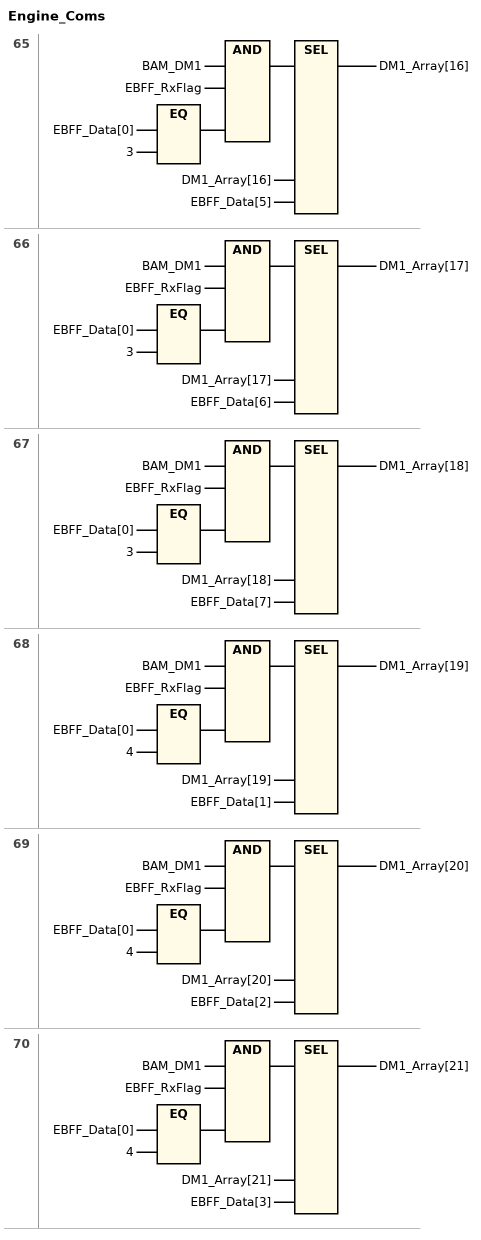
// NETWORK 65
DM1_Array[16] := SEL(BAM_DM1 AND EBFF_RxFlag AND EBFF_Data[0] = 3, DM1_Array[16], EBFF_Data[5]);

// NETWORK 66
DM1_Array[17] := SEL(BAM_DM1 AND EBFF_RxFlag AND EBFF_Data[0] = 3, DM1_Array[17], EBFF_Data[6]);

// NETWORK 67
DM1_Array[18] := SEL(BAM_DM1 AND EBFF_RxFlag AND EBFF_Data[0] = 3, DM1_Array[18], EBFF_Data[7]);

// NETWORK 68
DM1_Array[19] := SEL(BAM_DM1 AND EBFF_RxFlag AND EBFF_Data[0] = 4, DM1_Array[19], EBFF_Data[1]);

// NETWORK 69
DM1_Array[20] := SEL(BAM_DM1 AND EBFF_RxFlag AND EBFF_Data[0] = 4, DM1_Array[20], EBFF_Data[2]);

// NETWORK 70
DM1_Array[21] := SEL(BAM_DM1 AND EBFF_RxFlag AND EBFF_Data[0] = 4, DM1_Array[21], EBFF_Data[3]);

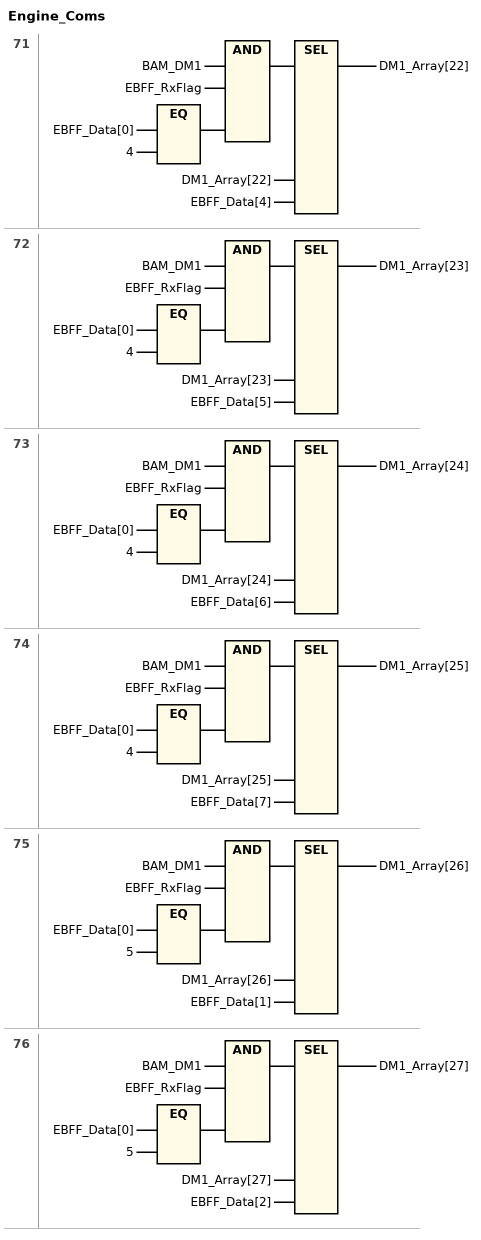
// NETWORK 71
DM1_Array[22] := SEL(BAM_DM1 AND EBFF_RxFlag AND EBFF_Data[0] = 4, DM1_Array[22], EBFF_Data[4]);

// NETWORK 72
DM1_Array[23] := SEL(BAM_DM1 AND EBFF_RxFlag AND EBFF_Data[0] = 4, DM1_Array[23], EBFF_Data[5]);

// NETWORK 73
DM1_Array[24] := SEL(BAM_DM1 AND EBFF_RxFlag AND EBFF_Data[0] = 4, DM1_Array[24], EBFF_Data[6]);

// NETWORK 74
DM1_Array[25] := SEL(BAM_DM1 AND EBFF_RxFlag AND EBFF_Data[0] = 4, DM1_Array[25], EBFF_Data[7]);

// NETWORK 75
DM1_Array[26] := SEL(BAM_DM1 AND EBFF_RxFlag AND EBFF_Data[0] = 5, DM1_Array[26], EBFF_Data[1]);

// NETWORK 76
DM1_Array[27] := SEL(BAM_DM1 AND EBFF_RxFlag AND EBFF_Data[0] = 5, DM1_Array[27], EBFF_Data[2]);

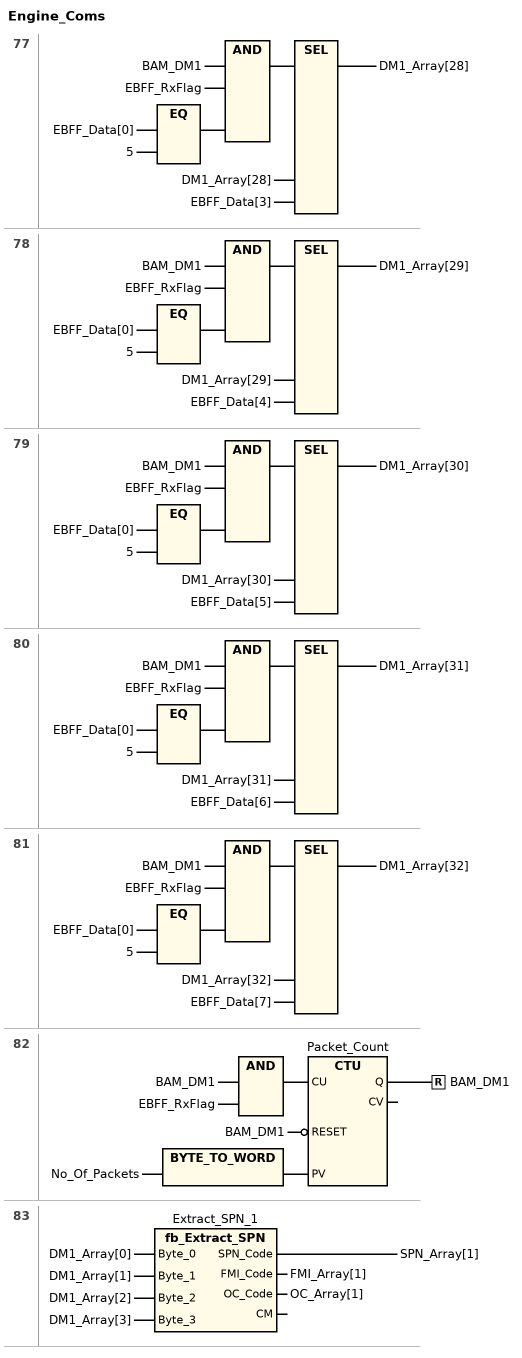
// NETWORK 77
DM1_Array[28] := SEL(BAM_DM1 AND EBFF_RxFlag AND EBFF_Data[0] = 5, DM1_Array[28], EBFF_Data[3]);

// NETWORK 78
DM1_Array[29] := SEL(BAM_DM1 AND EBFF_RxFlag AND EBFF_Data[0] = 5, DM1_Array[29], EBFF_Data[4]);

// NETWORK 79
DM1_Array[30] := SEL(BAM_DM1 AND EBFF_RxFlag AND EBFF_Data[0] = 5, DM1_Array[30], EBFF_Data[5]);

// NETWORK 80
DM1_Array[31] := SEL(BAM_DM1 AND EBFF_RxFlag AND EBFF_Data[0] = 5, DM1_Array[31], EBFF_Data[6]);

// NETWORK 81
DM1_Array[32] := SEL(BAM_DM1 AND EBFF_RxFlag AND EBFF_Data[0] = 5, DM1_Array[32], EBFF_Data[7]);

// NETWORK 82
Packet_Count(CU := BAM_DM1 AND EBFF_RxFlag, RESET := NOT BAM_DM1, PV := BYTE_TO_WORD(No_Of_Packets)); // CTU
BAM_DM1 R= Packet_Count.Q;

// NETWORK 83
Extract_SPN_1(
    Byte_0 := DM1_Array[0],
    Byte_1 := DM1_Array[1],
    Byte_2 := DM1_Array[2],
    Byte_3 := DM1_Array[3],
    FMI_Code => FMI_Array[1],
    OC_Code => OC_Array[1]); // fb_Extract_SPN
SPN_Array[1] := Extract_SPN_1.SPN_Code;

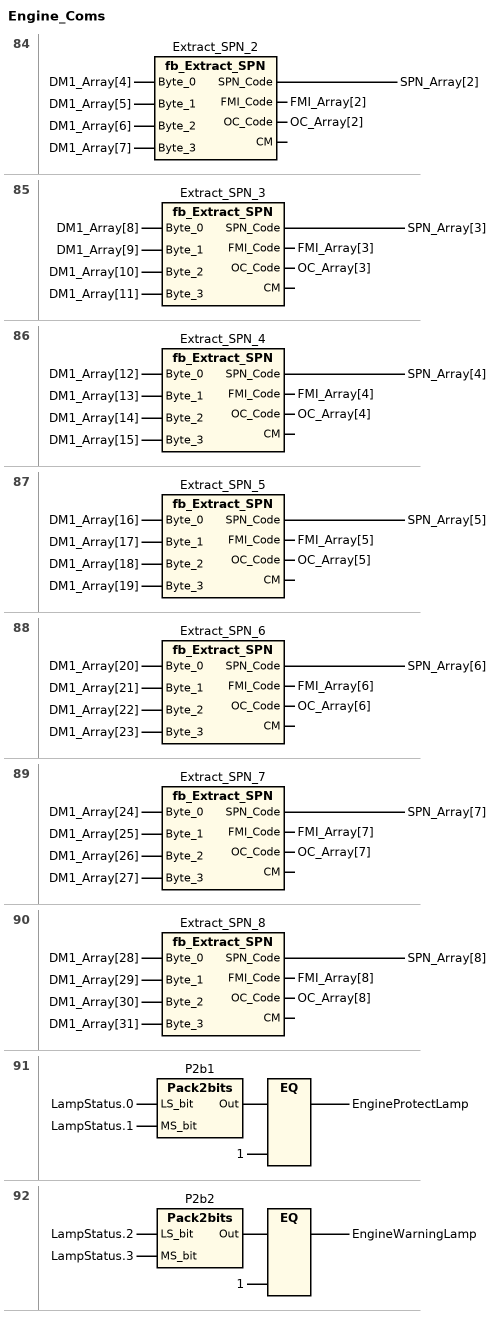
// NETWORK 84
Extract_SPN_2(
    Byte_0 := DM1_Array[4],
    Byte_1 := DM1_Array[5],
    Byte_2 := DM1_Array[6],
    Byte_3 := DM1_Array[7],
    FMI_Code => FMI_Array[2],
    OC_Code => OC_Array[2]); // fb_Extract_SPN
SPN_Array[2] := Extract_SPN_2.SPN_Code;

// NETWORK 85
Extract_SPN_3(
    Byte_0 := DM1_Array[8],
    Byte_1 := DM1_Array[9],
    Byte_2 := DM1_Array[10],
    Byte_3 := DM1_Array[11],
    FMI_Code => FMI_Array[3],
    OC_Code => OC_Array[3]); // fb_Extract_SPN
SPN_Array[3] := Extract_SPN_3.SPN_Code;

// NETWORK 86
Extract_SPN_4(
    Byte_0 := DM1_Array[12],
    Byte_1 := DM1_Array[13],
    Byte_2 := DM1_Array[14],
    Byte_3 := DM1_Array[15],
    FMI_Code => FMI_Array[4],
    OC_Code => OC_Array[4]); // fb_Extract_SPN
SPN_Array[4] := Extract_SPN_4.SPN_Code;

// NETWORK 87
Extract_SPN_5(
    Byte_0 := DM1_Array[16],
    Byte_1 := DM1_Array[17],
    Byte_2 := DM1_Array[18],
    Byte_3 := DM1_Array[19],
    FMI_Code => FMI_Array[5],
    OC_Code => OC_Array[5]); // fb_Extract_SPN
SPN_Array[5] := Extract_SPN_5.SPN_Code;

// NETWORK 88
Extract_SPN_6(
    Byte_0 := DM1_Array[20],
    Byte_1 := DM1_Array[21],
    Byte_2 := DM1_Array[22],
    Byte_3 := DM1_Array[23],
    FMI_Code => FMI_Array[6],
    OC_Code => OC_Array[6]); // fb_Extract_SPN
SPN_Array[6] := Extract_SPN_6.SPN_Code;

// NETWORK 89
Extract_SPN_7(
    Byte_0 := DM1_Array[24],
    Byte_1 := DM1_Array[25],
    Byte_2 := DM1_Array[26],
    Byte_3 := DM1_Array[27],
    FMI_Code => FMI_Array[7],
    OC_Code => OC_Array[7]); // fb_Extract_SPN
SPN_Array[7] := Extract_SPN_7.SPN_Code;

// NETWORK 90
Extract_SPN_8(
    Byte_0 := DM1_Array[28],
    Byte_1 := DM1_Array[29],
    Byte_2 := DM1_Array[30],
    Byte_3 := DM1_Array[31],
    FMI_Code => FMI_Array[8],
    OC_Code => OC_Array[8]); // fb_Extract_SPN
SPN_Array[8] := Extract_SPN_8.SPN_Code;

// NETWORK 91
P2b1(LS_bit := LampStatus.0, MS_bit := LampStatus.1); // Pack2bits
EngineProtectLamp := P2b1.Out = 1;

// NETWORK 92
P2b2(LS_bit := LampStatus.2, MS_bit := LampStatus.3); // Pack2bits
EngineWarningLamp := P2b2.Out = 1;

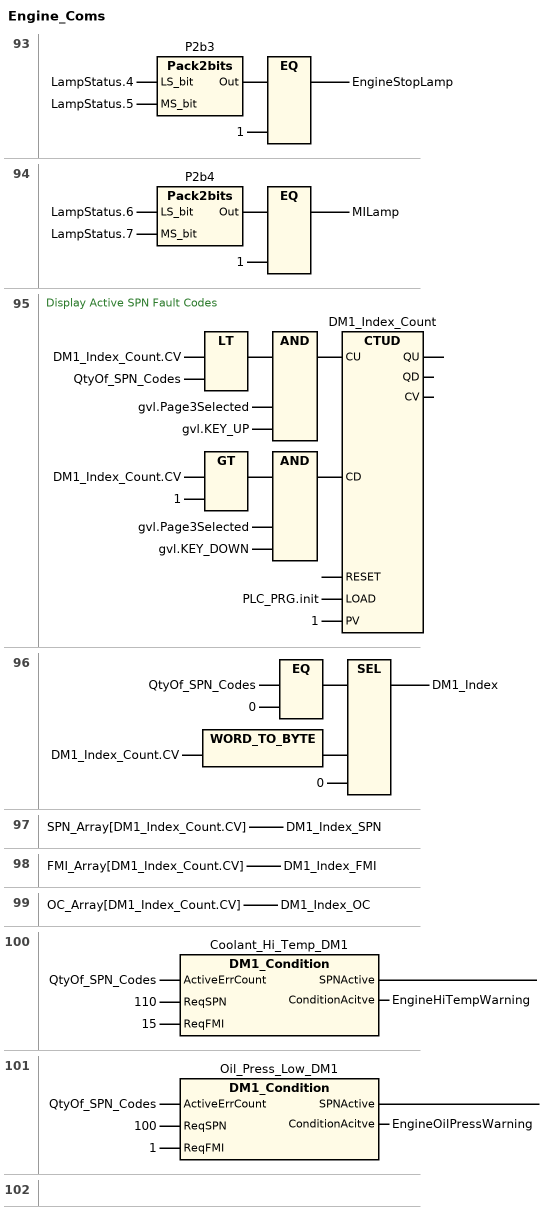
// NETWORK 93
P2b3(LS_bit := LampStatus.4, MS_bit := LampStatus.5); // Pack2bits
EngineStopLamp := P2b3.Out = 1;

// NETWORK 94
P2b4(LS_bit := LampStatus.6, MS_bit := LampStatus.7); // Pack2bits
MILamp := P2b4.Out = 1;

// NETWORK 95
// Display Active SPN Fault Codes
DM1_Index_Count(
    CU := DM1_Index_Count.CV < QtyOf_SPN_Codes AND gvl.Page3Selected AND gvl.KEY_UP,
    CD := DM1_Index_Count.CV > 1 AND gvl.Page3Selected AND gvl.KEY_DOWN,
    LOAD := PLC_PRG.init,
    PV := 1); // CTUD

// NETWORK 96
DM1_Index := SEL(QtyOf_SPN_Codes = 0, WORD_TO_BYTE(DM1_Index_Count.CV), 0);

// NETWORK 97
DM1_Index_SPN := SPN_Array[DM1_Index_Count.CV];

// NETWORK 98
DM1_Index_FMI := FMI_Array[DM1_Index_Count.CV];

// NETWORK 99
DM1_Index_OC := OC_Array[DM1_Index_Count.CV];

// NETWORK 100
Coolant_Hi_Temp_DM1(
    ActiveErrCount := QtyOf_SPN_Codes,
    ReqSPN := 110,
    ReqFMI := 15,
    ConditionAcitve => EngineHiTempWarning); // DM1_Condition

// NETWORK 101
Oil_Press_Low_DM1(
    ActiveErrCount := QtyOf_SPN_Codes,
    ReqSPN := 100,
    ReqFMI := 1,
    ConditionAcitve => EngineOilPressWarning); // DM1_Condition

// NETWORK 102

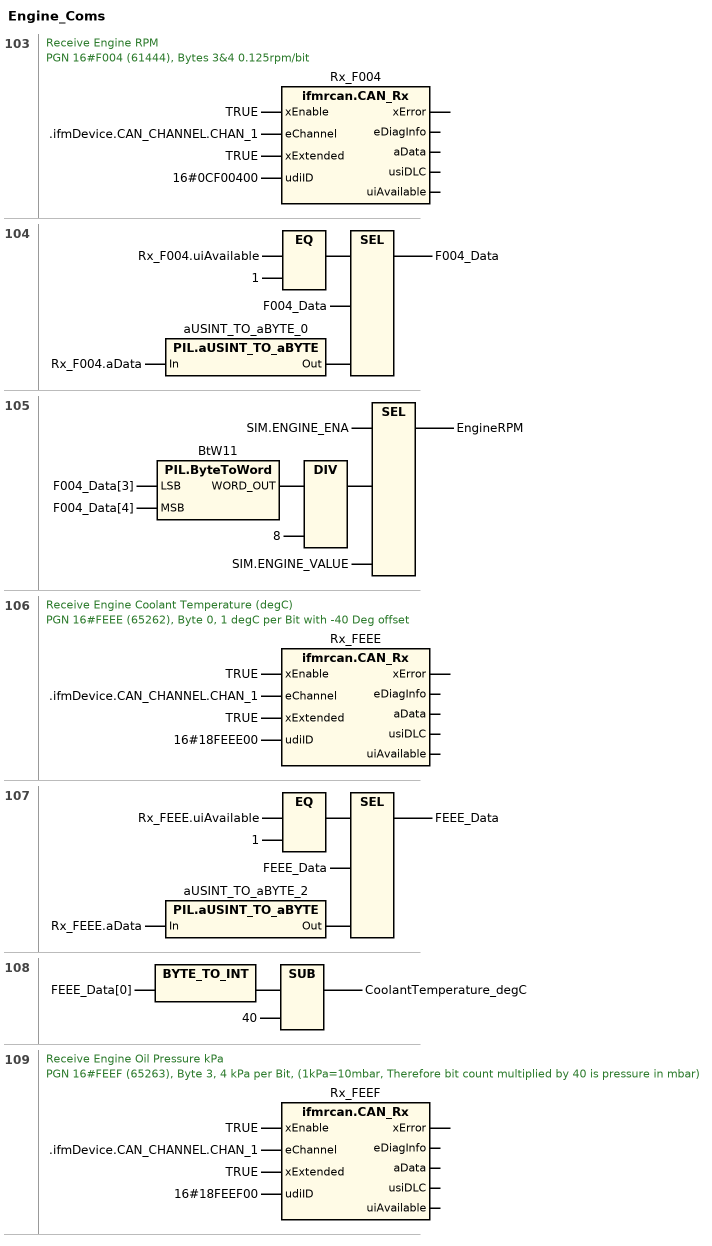
// NETWORK 103
// Receive Engine RPM
// PGN 16#F004 (61444), Bytes 3&4 0.125rpm/bit
Rx_F004(xEnable := TRUE, eChannel := .ifmDevice.CAN_CHANNEL.CHAN_1, xExtended := TRUE, udiID := 16#0CF00400); // ifmrcan.CAN_Rx

// NETWORK 104
aUSINT_TO_aBYTE_0(In := Rx_F004.aData); // PIL.aUSINT_TO_aBYTE
F004_Data := SEL(Rx_F004.uiAvailable = 1, F004_Data, aUSINT_TO_aBYTE_0.Out);

// NETWORK 105
BtW11(LSB := F004_Data[3], MSB := F004_Data[4]); // PIL.ByteToWord
EngineRPM := SEL(SIM.ENGINE_ENA, BtW11.WORD_OUT / 8, SIM.ENGINE_VALUE);

// NETWORK 106
// Receive Engine Coolant Temperature (degC)
// PGN 16#FEEE (65262), Byte 0, 1 degC per Bit with -40 Deg offset
Rx_FEEE(xEnable := TRUE, eChannel := .ifmDevice.CAN_CHANNEL.CHAN_1, xExtended := TRUE, udiID := 16#18FEEE00); // ifmrcan.CAN_Rx

// NETWORK 107
aUSINT_TO_aBYTE_2(In := Rx_FEEE.aData); // PIL.aUSINT_TO_aBYTE
FEEE_Data := SEL(Rx_FEEE.uiAvailable = 1, FEEE_Data, aUSINT_TO_aBYTE_2.Out);

// NETWORK 108
CoolantTemperature_degC := BYTE_TO_INT(FEEE_Data[0]) - 40;

// NETWORK 109
// Receive Engine Oil Pressure kPa
// PGN 16#FEEF (65263), Byte 3, 4 kPa per Bit, (1kPa=10mbar, Therefore bit count multiplied by 40 is pressure in mbar)
Rx_FEEF(xEnable := TRUE, eChannel := .ifmDevice.CAN_CHANNEL.CHAN_1, xExtended := TRUE, udiID := 16#18FEEF00); // ifmrcan.CAN_Rx

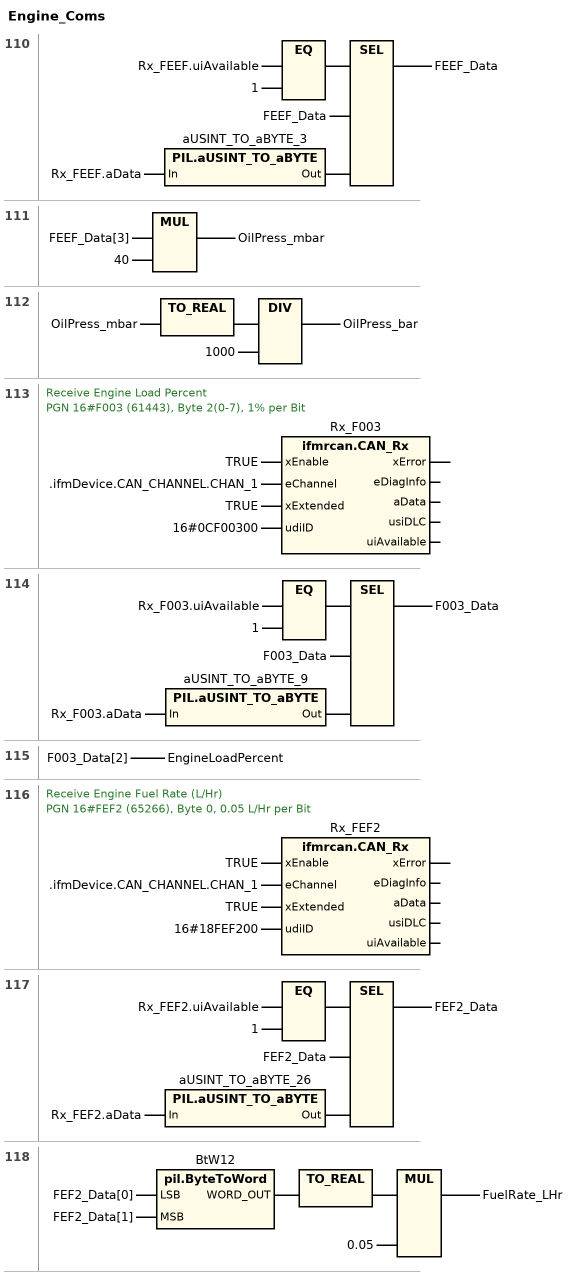
// NETWORK 110
aUSINT_TO_aBYTE_3(In := Rx_FEEF.aData); // PIL.aUSINT_TO_aBYTE
FEEF_Data := SEL(Rx_FEEF.uiAvailable = 1, FEEF_Data, aUSINT_TO_aBYTE_3.Out);

// NETWORK 111
OilPress_mbar := FEEF_Data[3] * 40;

// NETWORK 112
OilPress_bar := TO_REAL(OilPress_mbar) / 1000;

// NETWORK 113
// Receive Engine Load Percent
// PGN 16#F003 (61443), Byte 2(0-7), 1% per Bit
Rx_F003(xEnable := TRUE, eChannel := .ifmDevice.CAN_CHANNEL.CHAN_1, xExtended := TRUE, udiID := 16#0CF00300); // ifmrcan.CAN_Rx

// NETWORK 114
aUSINT_TO_aBYTE_9(In := Rx_F003.aData); // PIL.aUSINT_TO_aBYTE
F003_Data := SEL(Rx_F003.uiAvailable = 1, F003_Data, aUSINT_TO_aBYTE_9.Out);

// NETWORK 115
EngineLoadPercent := F003_Data[2];

// NETWORK 116
// Receive Engine Fuel Rate (L/Hr)
// PGN 16#FEF2 (65266), Byte 0, 0.05 L/Hr per Bit
Rx_FEF2(xEnable := TRUE, eChannel := .ifmDevice.CAN_CHANNEL.CHAN_1, xExtended := TRUE, udiID := 16#18FEF200); // ifmrcan.CAN_Rx

// NETWORK 117
aUSINT_TO_aBYTE_26(In := Rx_FEF2.aData); // PIL.aUSINT_TO_aBYTE
FEF2_Data := SEL(Rx_FEF2.uiAvailable = 1, FEF2_Data, aUSINT_TO_aBYTE_26.Out);

// NETWORK 118
BtW12(LSB := FEF2_Data[0], MSB := FEF2_Data[1]); // pil.ByteToWord
FuelRate_LHr := TO_REAL(BtW12.WORD_OUT) * 0.05;

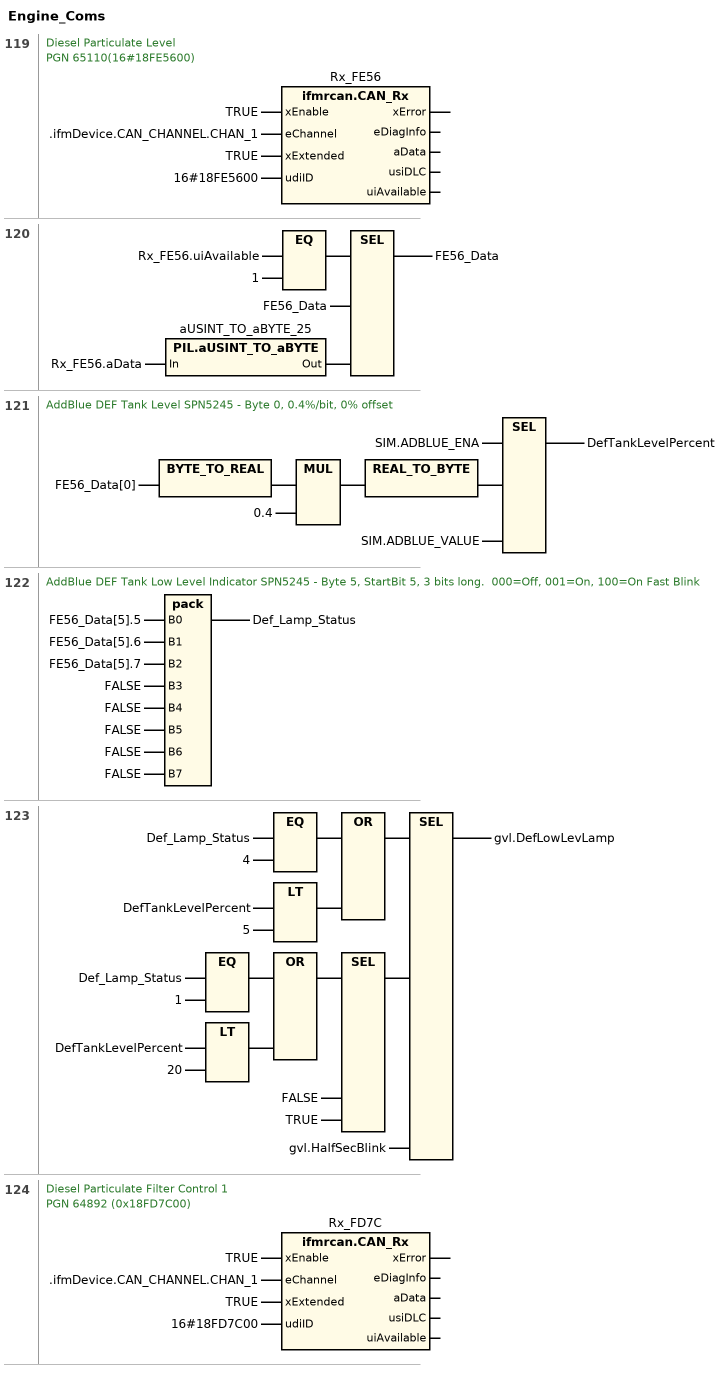
// NETWORK 119
// Diesel Particulate Level
// PGN 65110(16#18FE5600)
Rx_FE56(xEnable := TRUE, eChannel := .ifmDevice.CAN_CHANNEL.CHAN_1, xExtended := TRUE, udiID := 16#18FE5600); // ifmrcan.CAN_Rx

// NETWORK 120
aUSINT_TO_aBYTE_25(In := Rx_FE56.aData); // PIL.aUSINT_TO_aBYTE
FE56_Data := SEL(Rx_FE56.uiAvailable = 1, FE56_Data, aUSINT_TO_aBYTE_25.Out);

// NETWORK 121
// AddBlue DEF Tank Level SPN5245 - Byte 0, 0.4%/bit, 0% offset
DefTankLevelPercent := SEL(SIM.ADBLUE_ENA, REAL_TO_BYTE(BYTE_TO_REAL(FE56_Data[0]) * 0.4), SIM.ADBLUE_VALUE);

// NETWORK 122
// AddBlue DEF Tank Low Level Indicator SPN5245 - Byte 5, StartBit 5, 3 bits long.  000=Off, 001=On, 100=On Fast Blink
Def_Lamp_Status := pack(B0 := FE56_Data[5].5, B1 := FE56_Data[5].6, B2 := FE56_Data[5].7, B3 := FALSE, B4 := FALSE, B5 := FALSE, B6 := FALSE, B7 := FALSE);

// NETWORK 123
gvl.DefLowLevLamp := SEL(Def_Lamp_Status = 4 OR DefTankLevelPercent < 5, SEL(Def_Lamp_Status = 1 OR DefTankLevelPercent < 20, FALSE, TRUE), gvl.HalfSecBlink);

// NETWORK 124
// Diesel Particulate Filter Control 1
// PGN 64892 (0x18FD7C00)
Rx_FD7C(xEnable := TRUE, eChannel := .ifmDevice.CAN_CHANNEL.CHAN_1, xExtended := TRUE, udiID := 16#18FD7C00); // ifmrcan.CAN_Rx

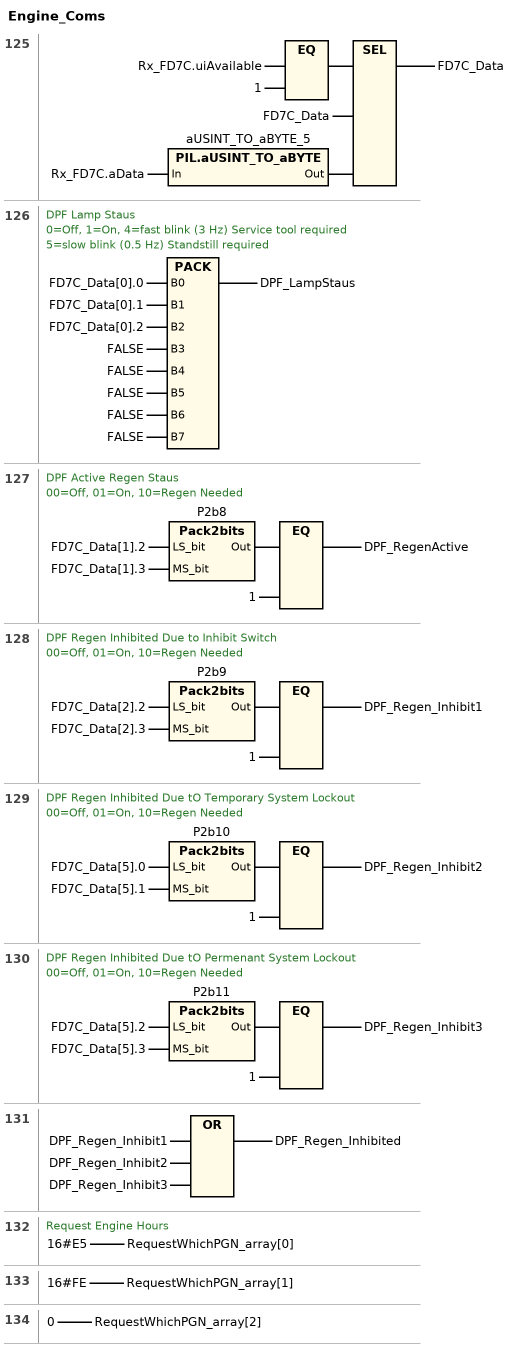
// NETWORK 125
aUSINT_TO_aBYTE_5(In := Rx_FD7C.aData); // PIL.aUSINT_TO_aBYTE
FD7C_Data := SEL(Rx_FD7C.uiAvailable = 1, FD7C_Data, aUSINT_TO_aBYTE_5.Out);

// NETWORK 126
// 					DPF Lamp Staus
// 0=Off, 1=On, 4=fast blink (3 Hz) Service tool required
// 5=slow blink (0.5 Hz) Standstill required
//
DPF_LampStaus := PACK(B0 := FD7C_Data[0].0, B1 := FD7C_Data[0].1, B2 := FD7C_Data[0].2, B3 := FALSE, B4 := FALSE, B5 := FALSE, B6 := FALSE, B7 := FALSE);

// NETWORK 127
// 					DPF Active Regen Staus
// 00=Off, 01=On, 10=Regen Needed
//
P2b8(LS_bit := FD7C_Data[1].2, MS_bit := FD7C_Data[1].3); // Pack2bits
DPF_RegenActive := P2b8.Out = 1;

// NETWORK 128
// 					DPF Regen Inhibited Due to Inhibit Switch
// 00=Off, 01=On, 10=Regen Needed
//
P2b9(LS_bit := FD7C_Data[2].2, MS_bit := FD7C_Data[2].3); // Pack2bits
DPF_Regen_Inhibit1 := P2b9.Out = 1;

// NETWORK 129
// 					DPF Regen Inhibited Due tO Temporary System Lockout
// 00=Off, 01=On, 10=Regen Needed
//
P2b10(LS_bit := FD7C_Data[5].0, MS_bit := FD7C_Data[5].1); // Pack2bits
DPF_Regen_Inhibit2 := P2b10.Out = 1;

// NETWORK 130
// 					DPF Regen Inhibited Due tO Permenant System Lockout
// 00=Off, 01=On, 10=Regen Needed
//
P2b11(LS_bit := FD7C_Data[5].2, MS_bit := FD7C_Data[5].3); // Pack2bits
DPF_Regen_Inhibit3 := P2b11.Out = 1;

// NETWORK 131
DPF_Regen_Inhibited := DPF_Regen_Inhibit1 OR DPF_Regen_Inhibit2 OR DPF_Regen_Inhibit3;

// NETWORK 132
// Request Engine Hours
RequestWhichPGN_array[0] := 16#E5;

// NETWORK 133
RequestWhichPGN_array[1] := 16#FE;

// NETWORK 134
RequestWhichPGN_array[2] := 0;

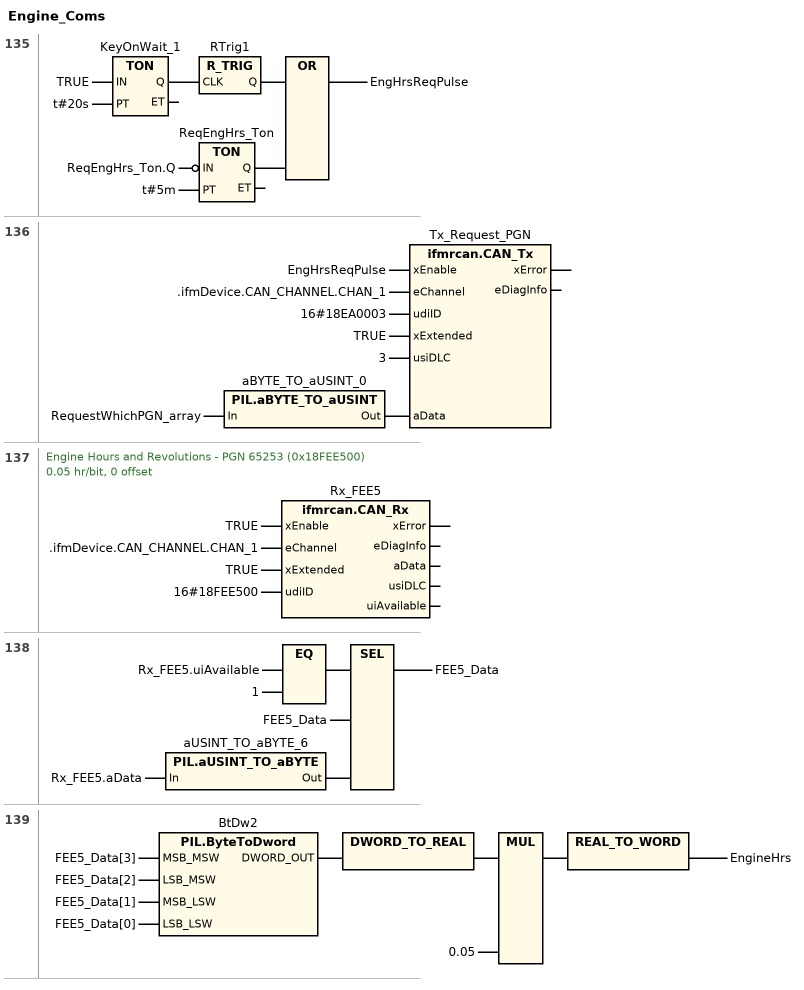
// NETWORK 135
KeyOnWait_1(IN := TRUE, PT := t#20s); // TON
RTrig1(CLK := KeyOnWait_1.Q); // R_TRIG
ReqEngHrs_Ton(IN := NOT ReqEngHrs_Ton.Q, PT := t#5m); // TON
EngHrsReqPulse := RTrig1.Q OR ReqEngHrs_Ton.Q;

// NETWORK 136
aBYTE_TO_aUSINT_0(In := RequestWhichPGN_array); // PIL.aBYTE_TO_aUSINT
Tx_Request_PGN(
    xEnable := EngHrsReqPulse,
    eChannel := .ifmDevice.CAN_CHANNEL.CHAN_1,
    udiID := 16#18EA0003,
    xExtended := TRUE,
    usiDLC := 3,
    aData := aBYTE_TO_aUSINT_0.Out); // ifmrcan.CAN_Tx

// NETWORK 137
// Engine Hours and Revolutions - PGN 65253 (0x18FEE500)
// 0.05 hr/bit, 0 offset
Rx_FEE5(xEnable := TRUE, eChannel := .ifmDevice.CAN_CHANNEL.CHAN_1, xExtended := TRUE, udiID := 16#18FEE500); // ifmrcan.CAN_Rx

// NETWORK 138
aUSINT_TO_aBYTE_6(In := Rx_FEE5.aData); // PIL.aUSINT_TO_aBYTE
FEE5_Data := SEL(Rx_FEE5.uiAvailable = 1, FEE5_Data, aUSINT_TO_aBYTE_6.Out);

// NETWORK 139
BtDw2(MSB_MSW := FEE5_Data[3], LSB_MSW := FEE5_Data[2], MSB_LSW := FEE5_Data[1], LSB_LSW := FEE5_Data[0]); // PIL.ByteToDword
EngineHrs := REAL_TO_WORD(DWORD_TO_REAL(BtDw2.DWORD_OUT) * 0.05);

END_PROGRAM

// StandardPLC/Application/CAN Comms/Engine Comms/CounterChecksum
FUNCTION_BLOCK CounterChecksum
VAR
	MessageCounter: BYTE;
	CheckSum: DWORD;
	MessageCheckSum: BYTE;
	ID_Low: BYTE;
	ID_midLow: BYTE;
	ID_midHigh: BYTE;
	ID_High: BYTE;
END_VAR
VAR_INPUT
	NewMessageTrig: BOOL;
	ID: DWORD;
END_VAR
VAR_OUTPUT
	Counter_ChecksumByte: BYTE;
END_VAR

ID_Low:=DWORD_TO_BYTE(ID);
ID_midLow:=DWORD_TO_BYTE(SHR(ID,8));
ID_midHigh:=DWORD_TO_BYTE(SHR(ID,16));
ID_High:=DWORD_TO_BYTE(SHR(ID,24));


IF NewMessageTrig=TRUE THEN MessageCounter:=MessageCounter+1;END_IF
IF MessageCounter>7 THEN MessageCounter:=0; END_IF

CheckSum:=Engine_Coms.Tx_TSC1.aData[0]+Engine_Coms.Tx_TSC1.aData[1]+Engine_Coms.Tx_TSC1.aData[2]+Engine_Coms.Tx_TSC1.aData[3]+
				Engine_Coms.Tx_TSC1.aData[4]+Engine_Coms.Tx_TSC1.aData[5]+Engine_Coms.Tx_TSC1.aData[6]+(MessageCounter AND 16#0F) + ID_Low + ID_midLow + ID_midHigh + ID_High;

MessageCheckSum:= DWORD_TO_BYTE((((SHR(CheckSum,6)) AND 16#03)+(SHR(CheckSum,3))+CheckSum) AND 16#07);

Counter_ChecksumByte:=SHL(MessageCheckSum,4)+MessageCounter;

END_FUNCTION_BLOCK

// StandardPLC/Application/CAN Comms/Engine Comms/fb_Extract_SPN
FUNCTION_BLOCK fb_Extract_SPN
VAR
	BtDW1: PIL.ByteToDword;
END_VAR
VAR_INPUT
	Byte_0: BYTE;
	Byte_1: BYTE;
	Byte_2: BYTE;
	Byte_3: BYTE;
END_VAR
VAR_OUTPUT
	SPN_Code: DWORD;
	FMI_Code: BYTE;
	OC_Code: BYTE;
	CM: BOOL;
END_VAR

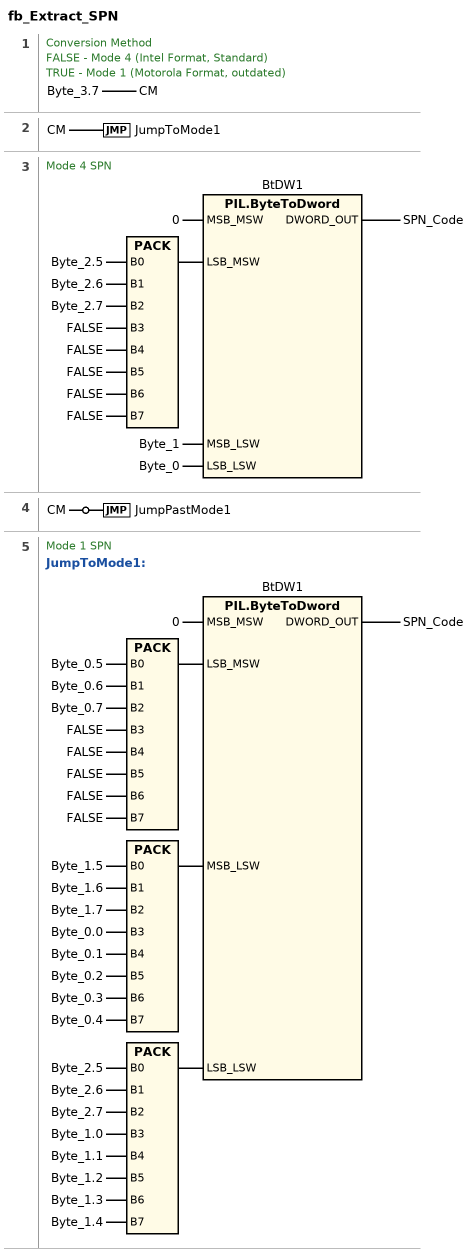
// NETWORK 1
// 					Conversion Method
// FALSE - Mode 4 (Intel Format, Standard)
// TRUE - Mode 1 (Motorola Format, outdated)
//
CM := Byte_3.7;

// NETWORK 2
IF CM THEN JMP JumpToMode1; END_IF

// NETWORK 3
// Mode 4 SPN
BtDW1(
    MSB_MSW := 0,
    LSB_MSW := PACK(B0 := Byte_2.5, B1 := Byte_2.6, B2 := Byte_2.7, B3 := FALSE, B4 := FALSE, B5 := FALSE, B6 := FALSE, B7 := FALSE),
    MSB_LSW := Byte_1,
    LSB_LSW := Byte_0); // PIL.ByteToDword
SPN_Code := BtDW1.DWORD_OUT;

// NETWORK 4
IF NOT CM THEN JMP JumpPastMode1; END_IF

// NETWORK 5
// Mode 1 SPN
JumpToMode1:
BtDW1(
    MSB_MSW := 0,
    LSB_MSW := PACK(B0 := Byte_0.5, B1 := Byte_0.6, B2 := Byte_0.7, B3 := FALSE, B4 := FALSE, B5 := FALSE, B6 := FALSE, B7 := FALSE),
    MSB_LSW := PACK(B0 := Byte_1.5, B1 := Byte_1.6, B2 := Byte_1.7, B3 := Byte_0.0, B4 := Byte_0.1, B5 := Byte_0.2, B6 := Byte_0.3, B7 := Byte_0.4),
    LSB_LSW := PACK(B0 := Byte_2.5, B1 := Byte_2.6, B2 := Byte_2.7, B3 := Byte_1.0, B4 := Byte_1.1, B5 := Byte_1.2, B6 := Byte_1.3, B7 := Byte_1.4)); // PIL.ByteToDword
SPN_Code := BtDW1.DWORD_OUT;

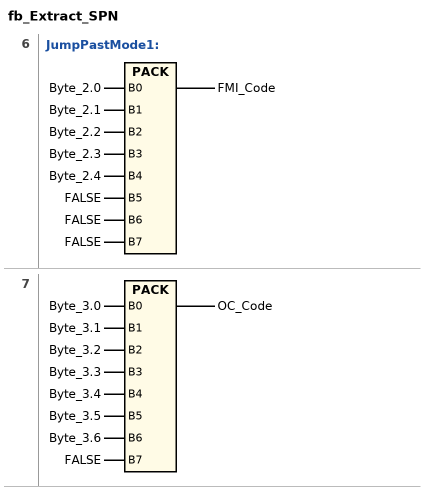
// NETWORK 6
JumpPastMode1:
FMI_Code := PACK(B0 := Byte_2.0, B1 := Byte_2.1, B2 := Byte_2.2, B3 := Byte_2.3, B4 := Byte_2.4, B5 := FALSE, B6 := FALSE, B7 := FALSE);

// NETWORK 7
OC_Code := PACK(B0 := Byte_3.0, B1 := Byte_3.1, B2 := Byte_3.2, B3 := Byte_3.3, B4 := Byte_3.4, B5 := Byte_3.5, B6 := Byte_3.6, B7 := FALSE);

END_FUNCTION_BLOCK

// StandardPLC/Application/CAN Comms/Engine Comms/Pack2bits
FUNCTION_BLOCK Pack2bits
VAR_INPUT
	LS_bit: BOOL;
	MS_bit: BOOL;
END_VAR
VAR_OUTPUT
	Out: BYTE;
END_VAR
VAR
END_VAR

IF LS_bit=TRUE THEN Out:=1; ELSE Out:=0; END_IF
IF MS_bit=TRUE THEN Out:=Out+2; ELSE Out:=Out; END_IF

END_FUNCTION_BLOCK

// StandardPLC/Application/CAN Comms/Engine Comms/DM1_Condition
FUNCTION_BLOCK DM1_Condition

(*Function block to look for an active SPN that is contained within the Error codes array [1..15]
The ConditionActive ouptut is used when you want to identify a SPN with a certain FMI
The SPNActive output is TRUE when the requested SPN is contained anywhere withing the array*)

VAR_INPUT
	ActiveErrCount: BYTE;
	ReqSPN: DWORD;
	ReqFMI: BYTE;
END_VAR
VAR_OUTPUT
	SPNActive: BOOL;
	ConditionAcitve: BOOL;
END_VAR
VAR
(*Temporary Variables*)
	SPNActive_1: BOOL;
	SPNActive_2: BOOL;
	SPNActive_3: BOOL;
	SPNActive_4: BOOL;
	SPNActive_5: BOOL;
	SPNActive_6: BOOL;
	SPNActive_7: BOOL;	(*  *)
	SPNActive_8: BOOL;	(*  *)
END_VAR
VAR // added by the converter: edge detectors and wires of the graphical bodies
    _w1, _w2, _w3, _w4, _w5, _w6, _w7, _w8 : BOOL;
END_VAR

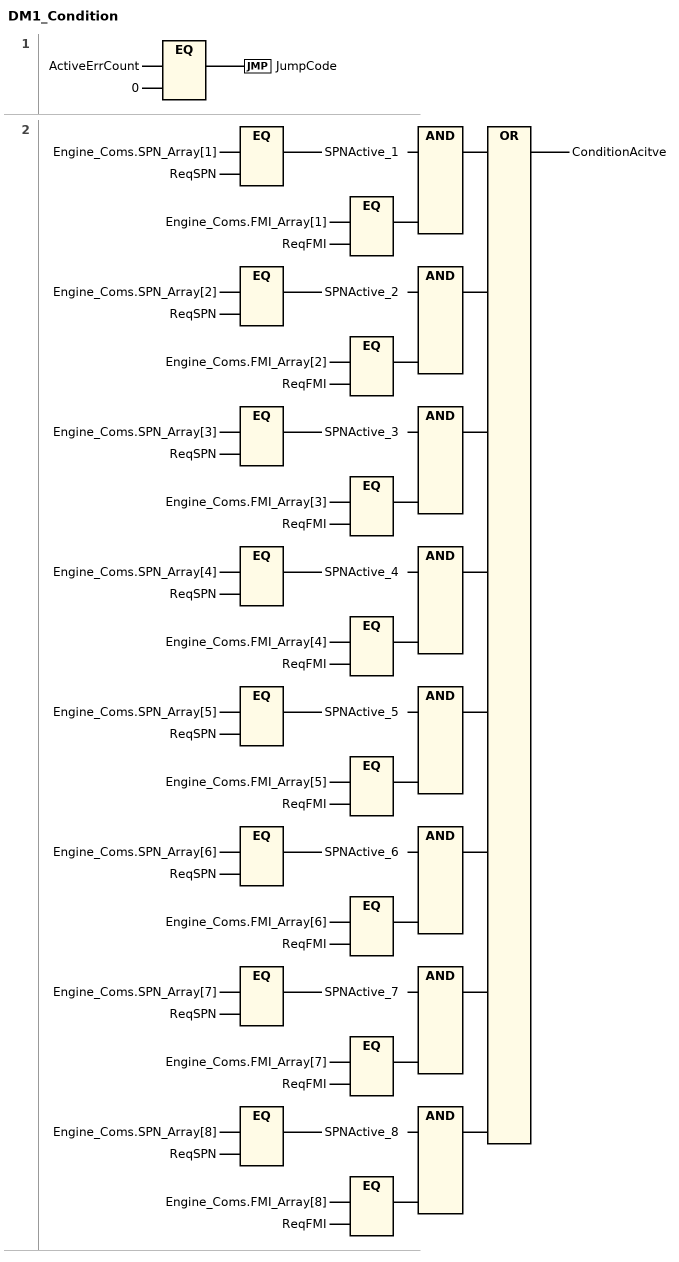
// NETWORK 1
IF ActiveErrCount = 0 THEN JMP JumpCode; END_IF

// NETWORK 2
_w1 := Engine_Coms.SPN_Array[1] = ReqSPN;
SPNActive_1 := _w1;
_w2 := Engine_Coms.SPN_Array[2] = ReqSPN;
SPNActive_2 := _w2;
_w3 := Engine_Coms.SPN_Array[3] = ReqSPN;
SPNActive_3 := _w3;
_w4 := Engine_Coms.SPN_Array[4] = ReqSPN;
SPNActive_4 := _w4;
_w5 := Engine_Coms.SPN_Array[5] = ReqSPN;
SPNActive_5 := _w5;
_w6 := Engine_Coms.SPN_Array[6] = ReqSPN;
SPNActive_6 := _w6;
_w7 := Engine_Coms.SPN_Array[7] = ReqSPN;
SPNActive_7 := _w7;
_w8 := Engine_Coms.SPN_Array[8] = ReqSPN;
SPNActive_8 := _w8;
ConditionAcitve := _w1 AND Engine_Coms.FMI_Array[1] = ReqFMI OR _w2 AND Engine_Coms.FMI_Array[2] = ReqFMI OR _w3 AND Engine_Coms.FMI_Array[3] = ReqFMI OR _w4 AND Engine_Coms.FMI_Array[4] = ReqFMI OR _w5 AND Engine_Coms.FMI_Array[5] = ReqFMI OR _w6 AND Engine_Coms.FMI_Array[6] = ReqFMI OR _w7 AND Engine_Coms.FMI_Array[7] = ReqFMI OR _w8 AND Engine_Coms.FMI_Array[8] = ReqFMI;

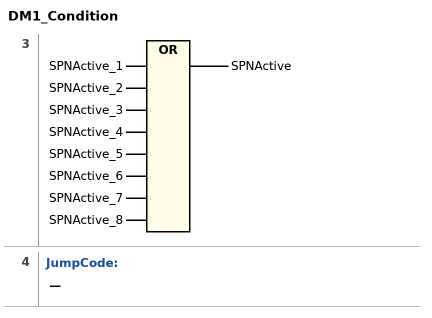
// NETWORK 3
SPNActive := SPNActive_1 OR SPNActive_2 OR SPNActive_3 OR SPNActive_4 OR SPNActive_5 OR SPNActive_6 OR SPNActive_7 OR SPNActive_8;

// NETWORK 4
JumpCode: ;

END_FUNCTION_BLOCK

// StandardPLC/Application/Set Points/SP_CountX1
FUNCTION_BLOCK SP_CountX1
VAR_INPUT
	Enable: BOOL;
	Value_In: INT;
	FastCount: BOOL;
	LowLim: INT;
	HiLim: INT;
END_VAR
VAR_OUTPUT
	Value_Out: INT;
END_VAR

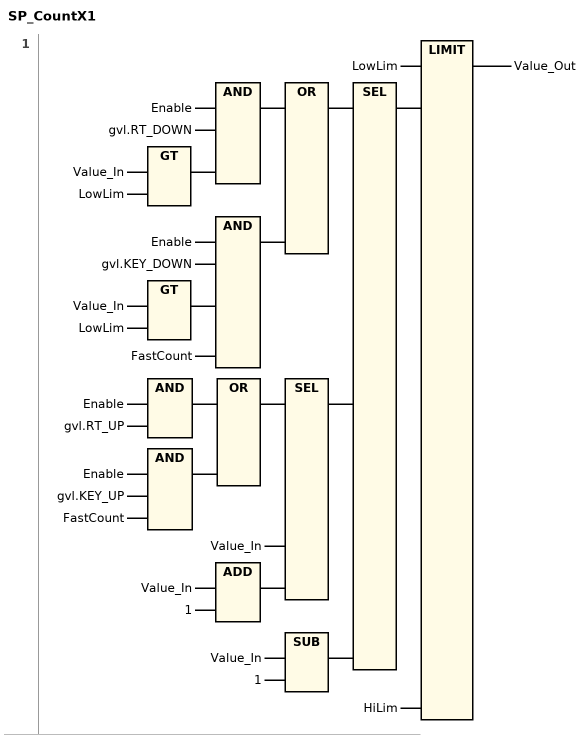
// NETWORK 1
Value_Out := LIMIT(LowLim, SEL(Enable AND gvl.RT_DOWN AND Value_In > LowLim OR Enable AND gvl.KEY_DOWN AND Value_In > LowLim AND FastCount, SEL(Enable AND gvl.RT_UP OR Enable AND gvl.KEY_UP AND FastCount, Value_In, Value_In + 1), Value_In - 1), HiLim);

END_FUNCTION_BLOCK

// StandardPLC/Application/Control/Tracking
PROGRAM Tracking
VAR
	RTrig1: R_TRIG;
	TrackingEnabled: PIL.PB_Toggle;
	WaitTon0: TON;
	Prestart: BOOL;
	BLINK_0: blink;
	AutoSequenceShutdown: BOOL;
	EngineRampDownSet: BOOL;
	EngineTo_1200rpm: BOOL;
	R_TRIG_0: r_TRig;
	WaitTon_1: TON;
END_VAR

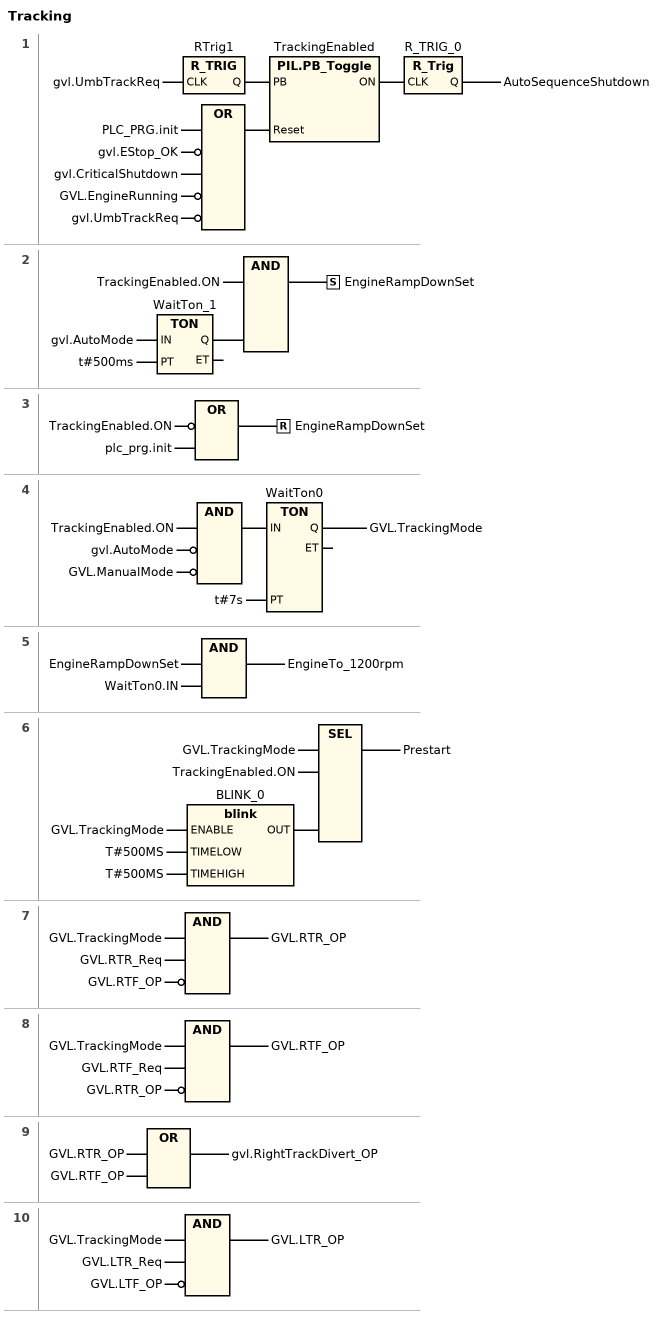
// NETWORK 1
RTrig1(CLK := gvl.UmbTrackReq); // R_TRIG
TrackingEnabled(PB := RTrig1.Q, Reset := PLC_PRG.init OR NOT gvl.EStop_OK OR gvl.CriticalShutdown OR NOT GVL.EngineRunning OR NOT gvl.UmbTrackReq); // PIL.PB_Toggle
R_TRIG_0(CLK := TrackingEnabled.ON); // R_Trig
AutoSequenceShutdown := R_TRIG_0.Q;

// NETWORK 2
WaitTon_1(IN := gvl.AutoMode, PT := t#500ms); // TON
EngineRampDownSet S= TrackingEnabled.ON AND WaitTon_1.Q;

// NETWORK 3
EngineRampDownSet R= NOT TrackingEnabled.ON OR plc_prg.init;

// NETWORK 4
WaitTon0(IN := TrackingEnabled.ON AND NOT gvl.AutoMode AND NOT GVL.ManualMode, PT := t#7s); // TON
GVL.TrackingMode := WaitTon0.Q;

// NETWORK 5
EngineTo_1200rpm := EngineRampDownSet AND WaitTon0.IN;

// NETWORK 6
BLINK_0(ENABLE := GVL.TrackingMode, TIMELOW := T#500MS, TIMEHIGH := T#500MS); // blink
Prestart := SEL(GVL.TrackingMode, TrackingEnabled.ON, BLINK_0.OUT);

// NETWORK 7
GVL.RTR_OP := GVL.TrackingMode AND GVL.RTR_Req AND NOT GVL.RTF_OP;

// NETWORK 8
GVL.RTF_OP := GVL.TrackingMode AND GVL.RTF_Req AND NOT GVL.RTR_OP;

// NETWORK 9
gvl.RightTrackDivert_OP := GVL.RTR_OP OR GVL.RTF_OP;

// NETWORK 10
GVL.LTR_OP := GVL.TrackingMode AND GVL.LTR_Req AND NOT GVL.LTF_OP;

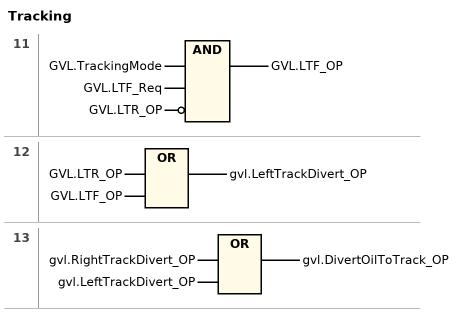
// NETWORK 11
GVL.LTF_OP := GVL.TrackingMode AND GVL.LTF_Req AND NOT GVL.LTR_OP;

// NETWORK 12
gvl.LeftTrackDivert_OP := GVL.LTR_OP OR GVL.LTF_OP;

// NETWORK 13
gvl.DivertOilToTrack_OP := gvl.RightTrackDivert_OP OR gvl.LeftTrackDivert_OP;

END_PROGRAM

// StandardPLC/Application/Control/Auto_Sequence
PROGRAM Auto_Sequence
VAR
	Blink1: BLINK;
	AutoStopMode: pil.PB_Toggle;
	AutoSequence: pil.PB_Toggle;
	PrestartTon: TON;
	Siren: BOOL;
	AutoStarting: BOOL;
	TailConv_PB: pil.PB_Toggle;
	WaitToStopTailConv: TON;
	TailConvOn: BOOL;
	WaitToStartSideConv: TON;
	WaitToStopSideConv: TON;
	SideConvOn: BOOL;
	SideConv_PB: pil.PB_Toggle;
	SideTransfer_PB: pil.PB_Toggle;
	WaitToStartSideTransfer: TON;
	WaitToStopSideTransfer: TON;
	SideTransferOn: BOOL;
	WaitToStartCollectConv: TON;
	WaitToStopCollectConv: TON;
	CollectConv_PB: pil.PB_Toggle;
	CollectConvOn: BOOL;
	WaitToStartDrum: TON;
	WaitToStopDrum: TON;
	Drum_PB: pil.PB_Toggle;
	DrumOn: BOOL;
	WaitToFeeder: TON;
	Feeder_PB: pil.PB_Toggle;
	FeederOn: BOOL;
	StartUpComplete: BOOL;
	F_TRIG_0: f_trig;
	F_TRIG_1: f_trig;
END_VAR
VAR RETAIN
END_VAR

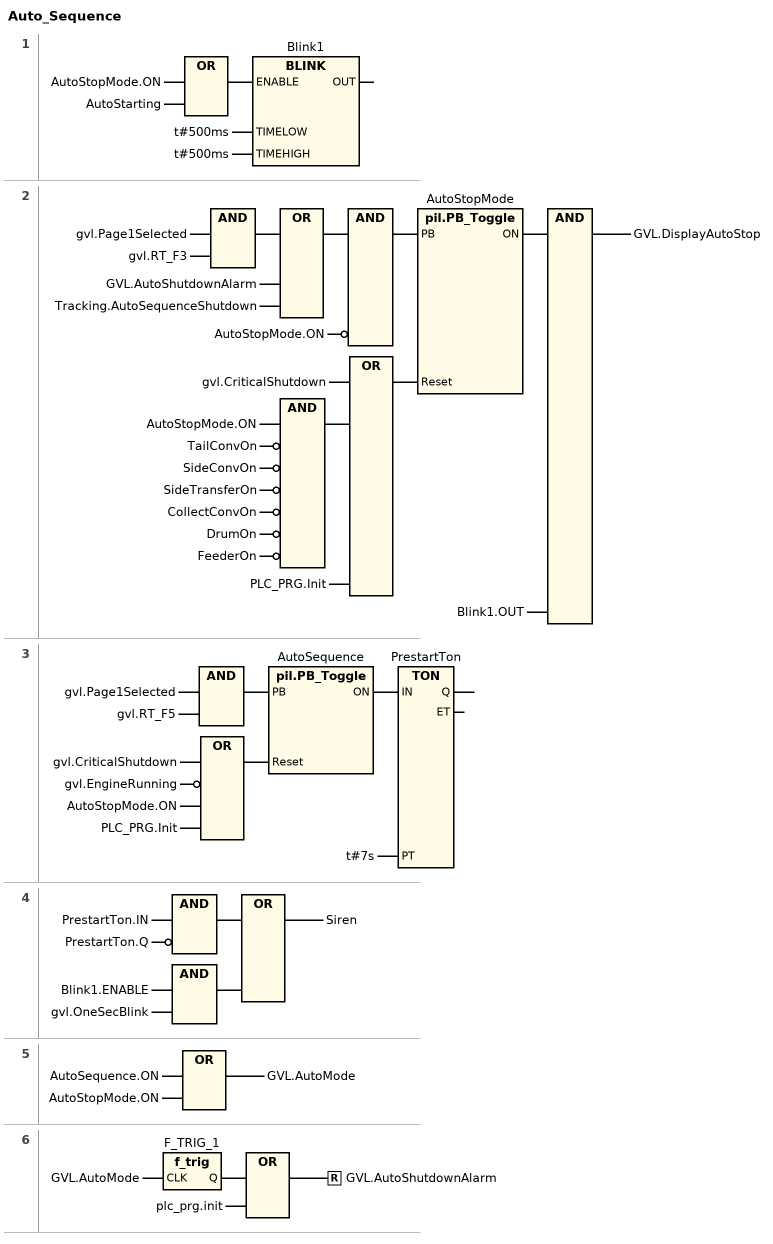
// NETWORK 1
Blink1(ENABLE := AutoStopMode.ON OR AutoStarting, TIMELOW := t#500ms, TIMEHIGH := t#500ms); // BLINK

// NETWORK 2
AutoStopMode(PB := (gvl.Page1Selected AND gvl.RT_F3 OR GVL.AutoShutdownAlarm OR Tracking.AutoSequenceShutdown) AND NOT AutoStopMode.ON, Reset := gvl.CriticalShutdown OR AutoStopMode.ON AND NOT TailConvOn AND NOT SideConvOn AND NOT SideTransferOn AND NOT CollectConvOn AND NOT DrumOn AND NOT FeederOn OR PLC_PRG.Init); // pil.PB_Toggle
GVL.DisplayAutoStop := AutoStopMode.ON AND Blink1.OUT;

// NETWORK 3
AutoSequence(PB := gvl.Page1Selected AND gvl.RT_F5, Reset := gvl.CriticalShutdown OR NOT gvl.EngineRunning OR AutoStopMode.ON OR PLC_PRG.Init); // pil.PB_Toggle
PrestartTon(IN := AutoSequence.ON, PT := t#7s); // TON

// NETWORK 4
Siren := PrestartTon.IN AND NOT PrestartTon.Q OR Blink1.ENABLE AND gvl.OneSecBlink;

// NETWORK 5
GVL.AutoMode := AutoSequence.ON OR AutoStopMode.ON;

// NETWORK 6
F_TRIG_1(CLK := GVL.AutoMode); // f_trig
GVL.AutoShutdownAlarm R= F_TRIG_1.Q OR plc_prg.init;

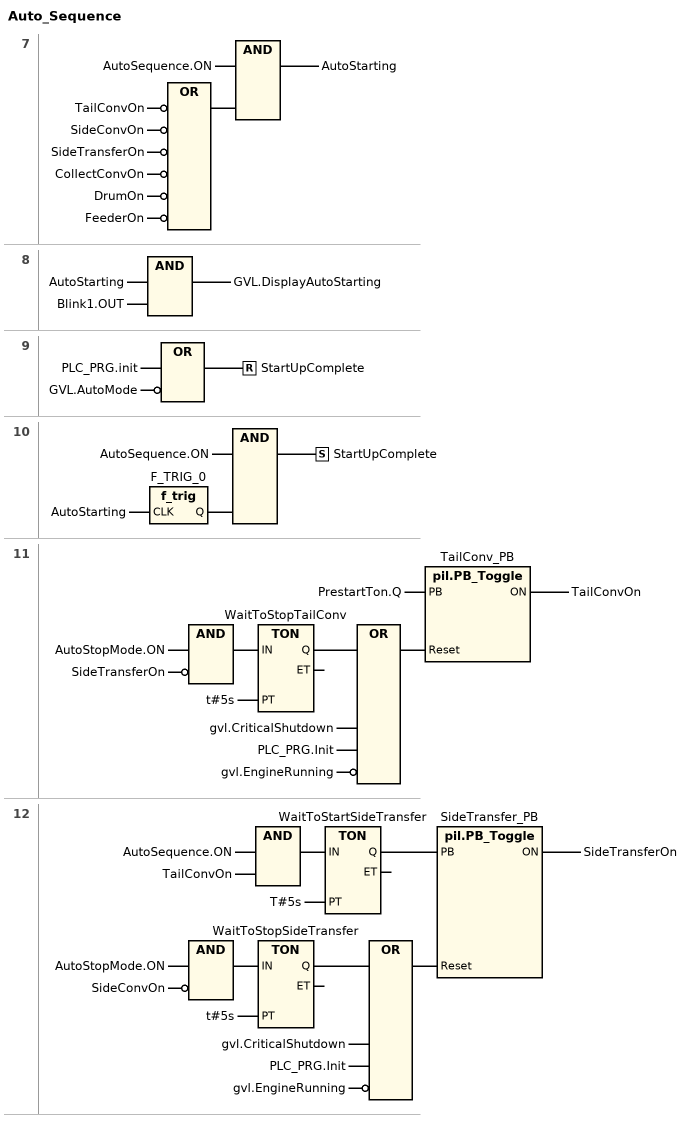
// NETWORK 7
AutoStarting := AutoSequence.ON AND (NOT TailConvOn OR NOT SideConvOn OR NOT SideTransferOn OR NOT CollectConvOn OR NOT DrumOn OR NOT FeederOn);

// NETWORK 8
GVL.DisplayAutoStarting := AutoStarting AND Blink1.OUT;

// NETWORK 9
StartUpComplete R= PLC_PRG.init OR NOT GVL.AutoMode;

// NETWORK 10
F_TRIG_0(CLK := AutoStarting); // f_trig
StartUpComplete S= AutoSequence.ON AND F_TRIG_0.Q;

// NETWORK 11
WaitToStopTailConv(IN := AutoStopMode.ON AND NOT SideTransferOn, PT := t#5s); // TON
TailConv_PB(PB := PrestartTon.Q, Reset := WaitToStopTailConv.Q OR gvl.CriticalShutdown OR PLC_PRG.Init OR NOT gvl.EngineRunning); // pil.PB_Toggle
TailConvOn := TailConv_PB.ON;

// NETWORK 12
WaitToStartSideTransfer(IN := AutoSequence.ON AND TailConvOn, PT := T#5s); // TON
WaitToStopSideTransfer(IN := AutoStopMode.ON AND NOT SideConvOn, PT := t#5s); // TON
SideTransfer_PB(PB := WaitToStartSideTransfer.Q, Reset := WaitToStopSideTransfer.Q OR gvl.CriticalShutdown OR PLC_PRG.Init OR NOT gvl.EngineRunning); // pil.PB_Toggle
SideTransferOn := SideTransfer_PB.ON;

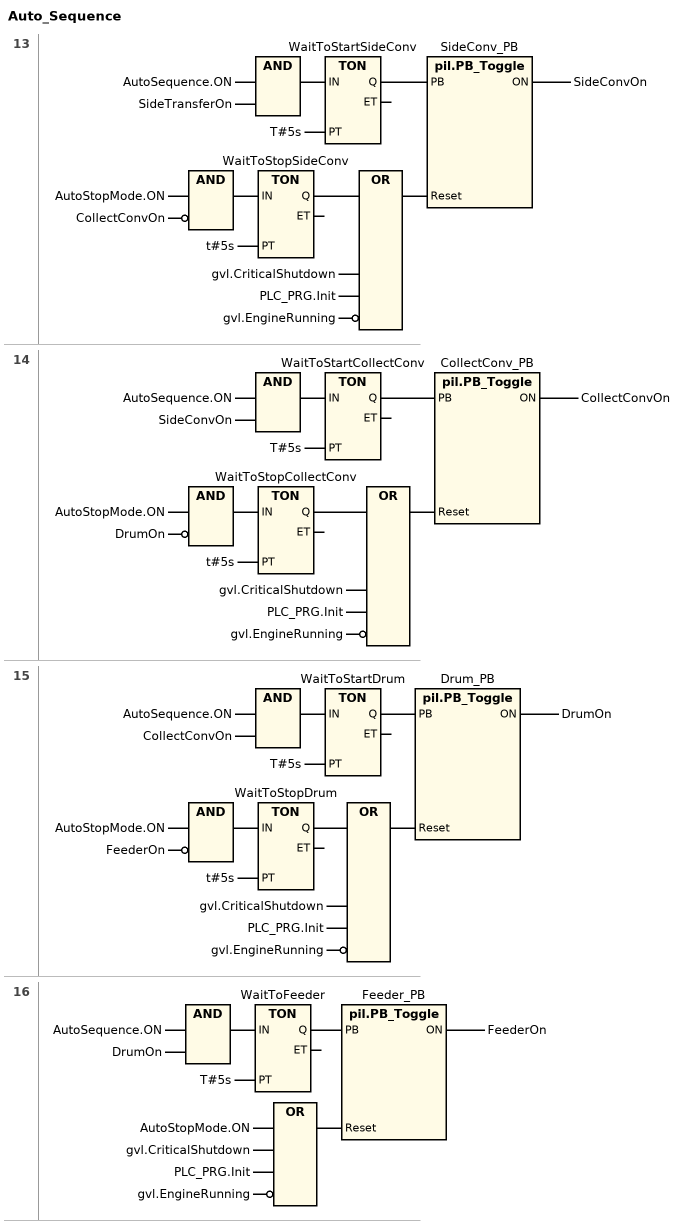
// NETWORK 13
WaitToStartSideConv(IN := AutoSequence.ON AND SideTransferOn, PT := T#5s); // TON
WaitToStopSideConv(IN := AutoStopMode.ON AND NOT CollectConvOn, PT := t#5s); // TON
SideConv_PB(PB := WaitToStartSideConv.Q, Reset := WaitToStopSideConv.Q OR gvl.CriticalShutdown OR PLC_PRG.Init OR NOT gvl.EngineRunning); // pil.PB_Toggle
SideConvOn := SideConv_PB.ON;

// NETWORK 14
WaitToStartCollectConv(IN := AutoSequence.ON AND SideConvOn, PT := T#5s); // TON
WaitToStopCollectConv(IN := AutoStopMode.ON AND NOT DrumOn, PT := t#5s); // TON
CollectConv_PB(PB := WaitToStartCollectConv.Q, Reset := WaitToStopCollectConv.Q OR gvl.CriticalShutdown OR PLC_PRG.Init OR NOT gvl.EngineRunning); // pil.PB_Toggle
CollectConvOn := CollectConv_PB.ON;

// NETWORK 15
WaitToStartDrum(IN := AutoSequence.ON AND CollectConvOn, PT := T#5s); // TON
WaitToStopDrum(IN := AutoStopMode.ON AND NOT FeederOn, PT := t#5s); // TON
Drum_PB(PB := WaitToStartDrum.Q, Reset := WaitToStopDrum.Q OR gvl.CriticalShutdown OR PLC_PRG.Init OR NOT gvl.EngineRunning); // pil.PB_Toggle
DrumOn := Drum_PB.ON;

// NETWORK 16
WaitToFeeder(IN := AutoSequence.ON AND DrumOn, PT := T#5s); // TON
Feeder_PB(PB := WaitToFeeder.Q, Reset := AutoStopMode.ON OR gvl.CriticalShutdown OR PLC_PRG.Init OR NOT gvl.EngineRunning); // pil.PB_Toggle
FeederOn := Feeder_PB.ON;

END_PROGRAM

// StandardPLC/Application/CAN Comms/CAN_COMS
  PROGRAM CAN_COMS
VAR
	EnableCAN0: ifmRCAN.CAN_Enable;
	Rx_100: ifmrcan.CAN_Rx;
	Rx100: ARRAY[0..7] OF BYTE;
	aUSINT_TO_aBYTE_1: PIL.aUSINT_TO_aBYTE;
	UP1: UNPACK;
	UP2: UNPACK;
	RTrig_F1: R_Trig;
	RTrig_F2: R_Trig;
	RTrig_F3: R_Trig;
	RTrig_F4: R_Trig;
	RTrig_F5: R_Trig;
	RTrig_F6: R_Trig;
	RTrig_Up: R_Trig;
	RTrig_Down: R_Trig;
	RTrig_Left: R_Trig;
	RTrig_Right: R_Trig;
	RTrig_OK: R_Trig;
	Rx_200: ifmrcan.CAN_Rx;
	aUSINT_TO_aBYTE_200: PIL.aUSINT_TO_aBYTE;
	Rx200: ARRAY[0..7] OF BYTE;
	Tx201: ifmrcan.CAN_Tx;
	Tx201_Ton: TON;
	UP3: UNPACK;
	Tx110_Ton: TON;
	Tx110: ifmrcan.CAN_Tx;
	HeartBeat: blink;
	Tx111_Ton: TON;
	Tx1110_Ton: BOOL;
	Tx111: ifmrcan.CAN_Tx;
	WtB1: pil.WordToByte;
	WtB2: pil.WordToByte;
	WtB3: pil.WordToByte;
	WtB4: pil.WordToByte;
	Tx112_Ton: TON;
	Tx112: ifmrcan.CAN_Tx;
	dWtB1: pil.DwordToByte;
	Tx113_Ton: TON;
	Tx113: ifmrcan.CAN_Tx;
	WtB5: pil.WordToByte;
	Tx114_Ton: TON;
	Tx114: ifmrcan.CAN_Tx;
	Tx115_Ton: TON;
	Tx115: ifmrcan.CAN_Tx;
	WtB6: pil.WordToByte;
	WtB7: pil.WordToByte;
	WtB8: pil.WordToByte;
	WtB9: pil.WordToByte;
	WtB10: pil.WordToByte;
	WtB11: pil.WordToByte;
	Tx116_Ton: TON;
	Tx116: ifmrcan.CAN_Tx;
	WtB12: pil.WordToByte;
	WtB13: pil.WordToByte;
	WtB14: pil.WordToByte;
	WtB15: pil.WordToByte;
	Tx117_Ton: TON;
	Tx117: ifmrcan.CAN_Tx;
	WtB16: pil.WordToByte;
	WtB17: pil.WordToByte;
	UP4: UNPACK;
	Tx118_Ton: TON;
	Tx118: ifmrcan.CAN_Tx;
	WtB18: pil.WordToByte;
END_VAR

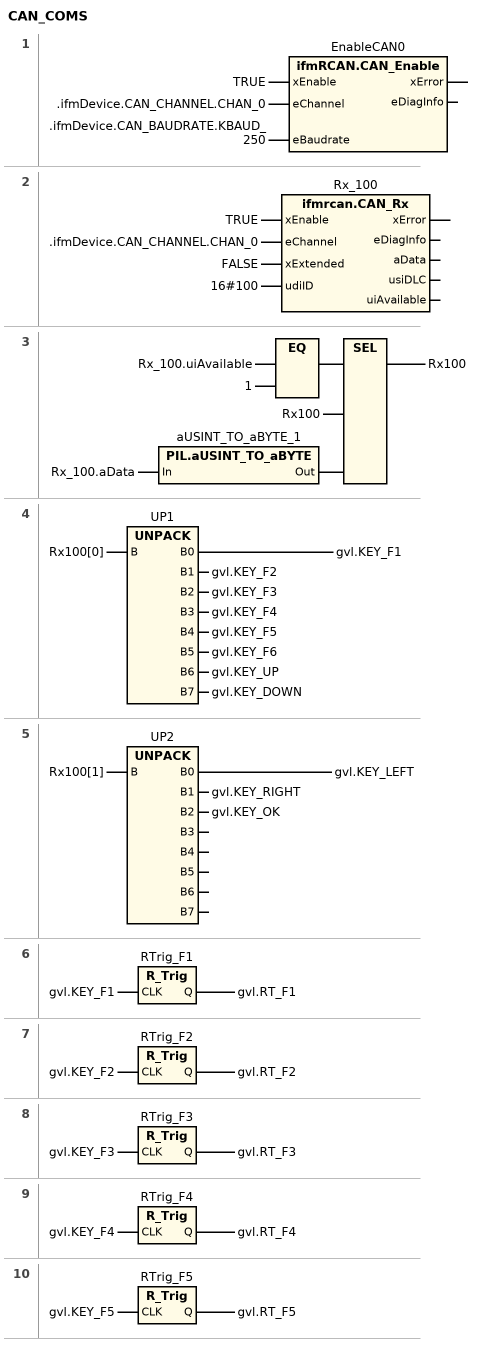
// NETWORK 1
EnableCAN0(
    xEnable := TRUE,
    eChannel := .ifmDevice.CAN_CHANNEL.CHAN_0,
    eBaudrate := .ifmDevice.CAN_BAUDRATE.KBAUD_250); // ifmRCAN.CAN_Enable

// NETWORK 2
Rx_100(xEnable := TRUE, eChannel := .ifmDevice.CAN_CHANNEL.CHAN_0, xExtended := FALSE, udiID := 16#100); // ifmrcan.CAN_Rx

// NETWORK 3
aUSINT_TO_aBYTE_1(In := Rx_100.aData); // PIL.aUSINT_TO_aBYTE
Rx100 := SEL(Rx_100.uiAvailable = 1, Rx100, aUSINT_TO_aBYTE_1.Out);

// NETWORK 4
UP1(
    B := Rx100[0],
    B1 => gvl.KEY_F2,
    B2 => gvl.KEY_F3,
    B3 => gvl.KEY_F4,
    B4 => gvl.KEY_F5,
    B5 => gvl.KEY_F6,
    B6 => gvl.KEY_UP,
    B7 => gvl.KEY_DOWN); // UNPACK
gvl.KEY_F1 := UP1.B0;

// NETWORK 5
UP2(B := Rx100[1], B1 => gvl.KEY_RIGHT, B2 => gvl.KEY_OK); // UNPACK
gvl.KEY_LEFT := UP2.B0;

// NETWORK 6
RTrig_F1(CLK := gvl.KEY_F1); // R_Trig
gvl.RT_F1 := RTrig_F1.Q;

// NETWORK 7
RTrig_F2(CLK := gvl.KEY_F2); // R_Trig
gvl.RT_F2 := RTrig_F2.Q;

// NETWORK 8
RTrig_F3(CLK := gvl.KEY_F3); // R_Trig
gvl.RT_F3 := RTrig_F3.Q;

// NETWORK 9
RTrig_F4(CLK := gvl.KEY_F4); // R_Trig
gvl.RT_F4 := RTrig_F4.Q;

// NETWORK 10
RTrig_F5(CLK := gvl.KEY_F5); // R_Trig
gvl.RT_F5 := RTrig_F5.Q;

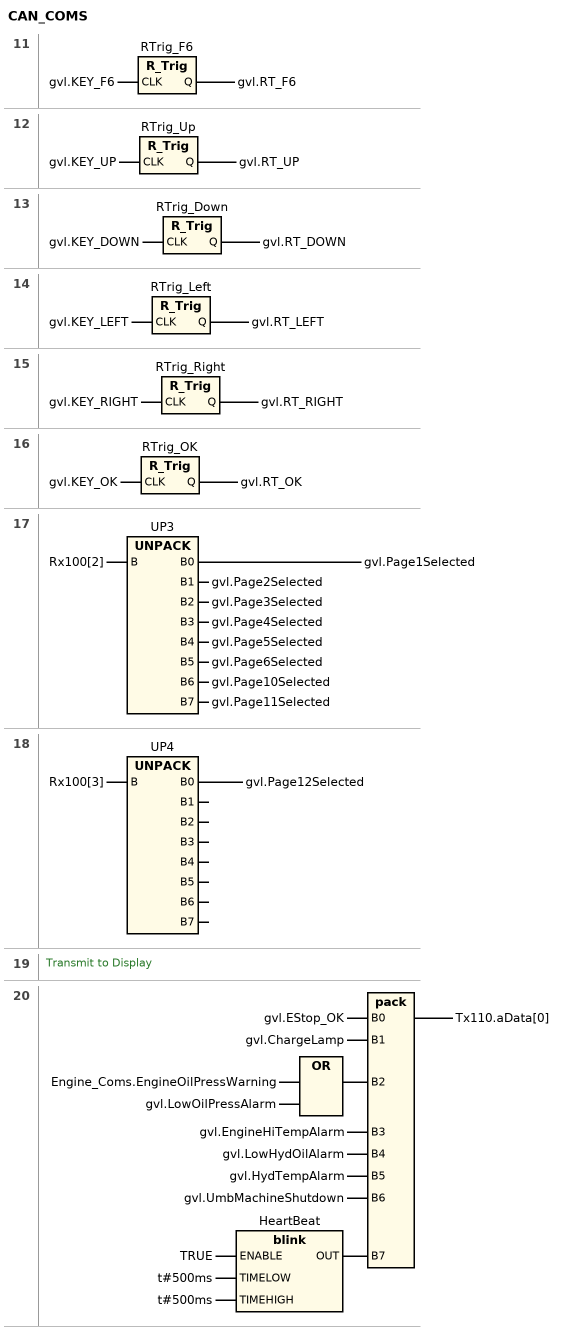
// NETWORK 11
RTrig_F6(CLK := gvl.KEY_F6); // R_Trig
gvl.RT_F6 := RTrig_F6.Q;

// NETWORK 12
RTrig_Up(CLK := gvl.KEY_UP); // R_Trig
gvl.RT_UP := RTrig_Up.Q;

// NETWORK 13
RTrig_Down(CLK := gvl.KEY_DOWN); // R_Trig
gvl.RT_DOWN := RTrig_Down.Q;

// NETWORK 14
RTrig_Left(CLK := gvl.KEY_LEFT); // R_Trig
gvl.RT_LEFT := RTrig_Left.Q;

// NETWORK 15
RTrig_Right(CLK := gvl.KEY_RIGHT); // R_Trig
gvl.RT_RIGHT := RTrig_Right.Q;

// NETWORK 16
RTrig_OK(CLK := gvl.KEY_OK); // R_Trig
gvl.RT_OK := RTrig_OK.Q;

// NETWORK 17
UP3(
    B := Rx100[2],
    B1 => gvl.Page2Selected,
    B2 => gvl.Page3Selected,
    B3 => gvl.Page4Selected,
    B4 => gvl.Page5Selected,
    B5 => gvl.Page6Selected,
    B6 => gvl.Page10Selected,
    B7 => gvl.Page11Selected); // UNPACK
gvl.Page1Selected := UP3.B0;

// NETWORK 18
UP4(B := Rx100[3]); // UNPACK
gvl.Page12Selected := UP4.B0;

// NETWORK 19
// Transmit to Display

// NETWORK 20
HeartBeat(ENABLE := TRUE, TIMELOW := t#500ms, TIMEHIGH := t#500ms); // blink
Tx110.aData[0] := pack(B0 := gvl.EStop_OK, B1 := gvl.ChargeLamp, B2 := Engine_Coms.EngineOilPressWarning OR gvl.LowOilPressAlarm, B3 := gvl.EngineHiTempAlarm, B4 := gvl.LowHydOilAlarm, B5 := gvl.HydTempAlarm, B6 := gvl.UmbMachineShutdown, B7 := HeartBeat.OUT);

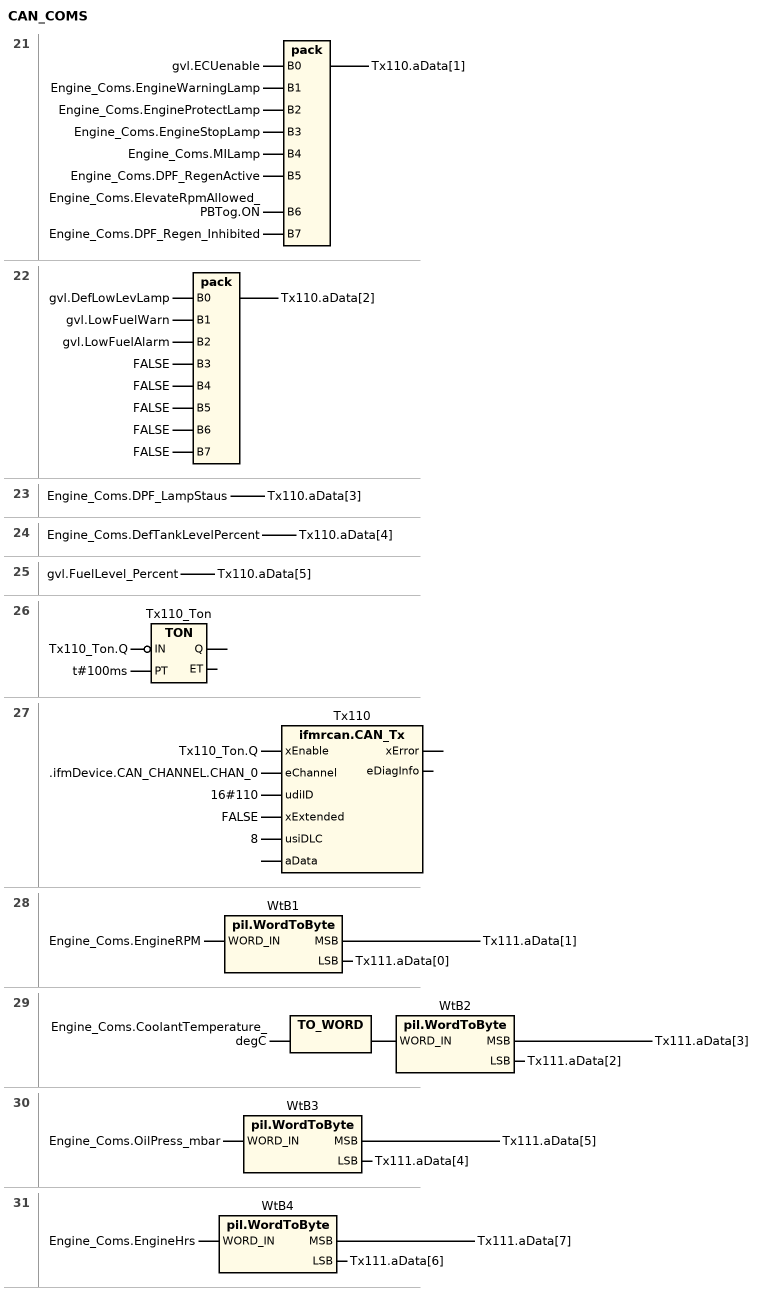
// NETWORK 21
Tx110.aData[1] := pack(B0 := gvl.ECUenable, B1 := Engine_Coms.EngineWarningLamp, B2 := Engine_Coms.EngineProtectLamp, B3 := Engine_Coms.EngineStopLamp, B4 := Engine_Coms.MILamp, B5 := Engine_Coms.DPF_RegenActive, B6 := Engine_Coms.ElevateRpmAllowed_PBTog.ON, B7 := Engine_Coms.DPF_Regen_Inhibited);

// NETWORK 22
Tx110.aData[2] := pack(B0 := gvl.DefLowLevLamp, B1 := gvl.LowFuelWarn, B2 := gvl.LowFuelAlarm, B3 := FALSE, B4 := FALSE, B5 := FALSE, B6 := FALSE, B7 := FALSE);

// NETWORK 23
Tx110.aData[3] := Engine_Coms.DPF_LampStaus;

// NETWORK 24
Tx110.aData[4] := Engine_Coms.DefTankLevelPercent;

// NETWORK 25
Tx110.aData[5] := gvl.FuelLevel_Percent;

// NETWORK 26
Tx110_Ton(IN := NOT Tx110_Ton.Q, PT := t#100ms); // TON

// NETWORK 27
Tx110(
    xEnable := Tx110_Ton.Q,
    eChannel := .ifmDevice.CAN_CHANNEL.CHAN_0,
    udiID := 16#110,
    xExtended := FALSE,
    usiDLC := 8); // ifmrcan.CAN_Tx

// NETWORK 28
WtB1(WORD_IN := Engine_Coms.EngineRPM, LSB => Tx111.aData[0]); // pil.WordToByte
Tx111.aData[1] := WtB1.MSB;

// NETWORK 29
WtB2(WORD_IN := TO_WORD(Engine_Coms.CoolantTemperature_degC), LSB => Tx111.aData[2]); // pil.WordToByte
Tx111.aData[3] := WtB2.MSB;

// NETWORK 30
WtB3(WORD_IN := Engine_Coms.OilPress_mbar, LSB => Tx111.aData[4]); // pil.WordToByte
Tx111.aData[5] := WtB3.MSB;

// NETWORK 31
WtB4(WORD_IN := Engine_Coms.EngineHrs, LSB => Tx111.aData[6]); // pil.WordToByte
Tx111.aData[7] := WtB4.MSB;

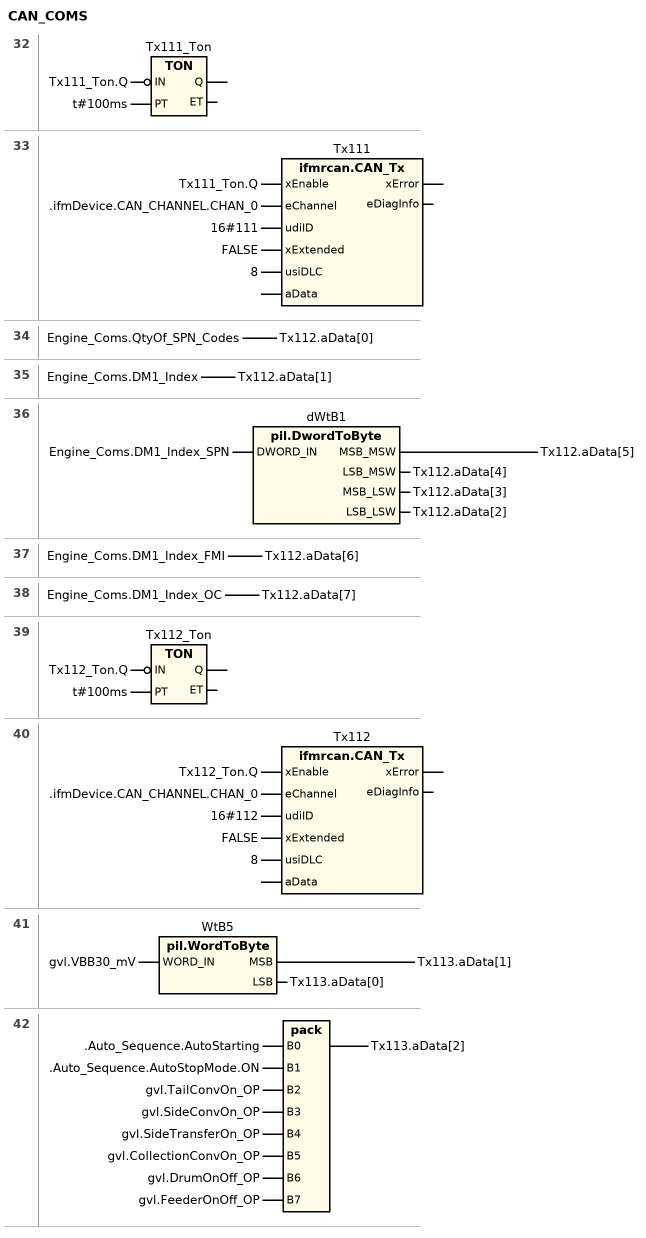
// NETWORK 32
Tx111_Ton(IN := NOT Tx111_Ton.Q, PT := t#100ms); // TON

// NETWORK 33
Tx111(
    xEnable := Tx111_Ton.Q,
    eChannel := .ifmDevice.CAN_CHANNEL.CHAN_0,
    udiID := 16#111,
    xExtended := FALSE,
    usiDLC := 8); // ifmrcan.CAN_Tx

// NETWORK 34
Tx112.aData[0] := Engine_Coms.QtyOf_SPN_Codes;

// NETWORK 35
Tx112.aData[1] := Engine_Coms.DM1_Index;

// NETWORK 36
dWtB1(
    DWORD_IN := Engine_Coms.DM1_Index_SPN,
    LSB_MSW => Tx112.aData[4],
    MSB_LSW => Tx112.aData[3],
    LSB_LSW => Tx112.aData[2]); // pil.DwordToByte
Tx112.aData[5] := dWtB1.MSB_MSW;

// NETWORK 37
Tx112.aData[6] := Engine_Coms.DM1_Index_FMI;

// NETWORK 38
Tx112.aData[7] := Engine_Coms.DM1_Index_OC;

// NETWORK 39
Tx112_Ton(IN := NOT Tx112_Ton.Q, PT := t#100ms); // TON

// NETWORK 40
Tx112(
    xEnable := Tx112_Ton.Q,
    eChannel := .ifmDevice.CAN_CHANNEL.CHAN_0,
    udiID := 16#112,
    xExtended := FALSE,
    usiDLC := 8); // ifmrcan.CAN_Tx

// NETWORK 41
WtB5(WORD_IN := gvl.VBB30_mV, LSB => Tx113.aData[0]); // pil.WordToByte
Tx113.aData[1] := WtB5.MSB;

// NETWORK 42
Tx113.aData[2] := pack(B0 := .Auto_Sequence.AutoStarting, B1 := .Auto_Sequence.AutoStopMode.ON, B2 := gvl.TailConvOn_OP, B3 := gvl.SideConvOn_OP, B4 := gvl.SideTransferOn_OP, B5 := gvl.CollectionConvOn_OP, B6 := gvl.DrumOnOff_OP, B7 := gvl.FeederOnOff_OP);

